TYPE "MES_Msg_Receive_Topic2xx_Err"
VERSION : 0.1
// Block: MES_Msg_Receive_Topic2xx_Err
   STRUCT
      Recive_MSG200 : "MES_Err_&_Msg";
      Recive_MSG210 : "MES_Err_&_Msg";
      Recive_MSG212 : "MES_Err_&_Msg";
      Send_MSG201_Follow_MSG200 : "MES_Err_&_Msg";
      Send_MSG211_Follow_MSG210 : "MES_Err_&_Msg";
   END_STRUCT;

END_TYPE
